// TIA Portal project "Mühürleme Devresi Uygulaması" (V18)

(* hardware
DEVICE "S7-1200 station_1"  S7-1200 Station
   slot 0: "Rack_0"  S7-1200 Rack  Rack  V1.0
   slot 1: "PLC_1"  CPU 1214C AC/DC/Rly  6ES7 214-1BG40-0XB0  V4.6
*)

// ===== PLC "PLC_1"  CPU 1214C AC/DC/Rly =====

VAR_GLOBAL   // PLC tag table "Default tag table"
   "Stop" AT %I0.0 : Bool;
   "Start_1" AT %I0.1 : Bool;
   "Start_2" AT %I0.2 : Bool;
   "Motor_1" AT %Q0.0 : Bool;
   "Start_3" AT %I0.3 : Bool;
   "Motor_2" AT %Q0.1 : Bool;
   "Motor_3" AT %Q0.2 : Bool;
END_VAR

ORGANIZATION_BLOCK "Main"   // OB1, LAD, ProgramCycle
TITLE = "Main Program Sweep (Cycle)"
{ S7_Optimized_Access := 'TRUE' }
VERSION : 0.1
   VAR_INPUT
      Initial_Call : Bool;   // Initial call of this OB
      Remanence : Bool;   // =True, if remanent data are available
   END_VAR
BEGIN

REGION Network 1
   // Start butonuna basıldığında çıkış rölesi çekecek. Butonu bıraktığımızda çıkış rölesi çekili kalacaktır. Stop butonuna basıldığında röle bırakacaktır. Motor aşırı akım çektiğinde motorun enerjisi kesilir.
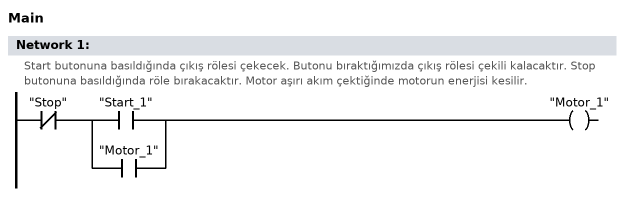
   RUNG wire#powerrail
      I_Contact( "Stop" )
      wire#w1
      Contact( "Start_1" )
      wire#w2
      Coil( "Motor_1" )
   END_RUNG
   RUNG wire#w1
      Contact( "Motor_1" )
   END_RUNG wire#w2
   // the same network as SCL:
   "Motor_1" := NOT "Stop" AND ("Start_1" OR "Motor_1");
END_REGION
END_ORGANIZATION_BLOCK